// TIA Portal V21 export
DATA_BLOCK "LayoutPercorsi"   // DB2
{ S7_Optimized_Access := 'TRUE' }
// stored: MemoryReserve 100
   VAR
      PercorsoDa : Struct
         SerbatoioProdotto : Int := 5;
         PompaMono : Int := 5;
         ContropressioneUscitaMono : Int := 0;
         PompaPistoni : Int := 5;
         Sterilizzazione : Int := 5;
         RicicloLavoroASostatore : Int := 5;
         RicicloLavoroASottoRaffreddatore : Int := 0;
         Sostatore : Int := 5;
         Raffreddatore : Int := 5;
         IngressoAcidoCamiciaRaffreddatore : Int := 0;
         IngressoH20RaffreddamentoVersoMod : Int := 1;
         IngressoH20RaffreddamentoVersoSottoRaffredda : Int := 1;
         DevioAcidoCamiciaRaffreddatore : Int := 0;
         RitornoProdottoVersoValvolaVapInSterilizzazione : Int := 0;
         QCI : Int := 5;
         IngressoProdottoInVasca : Int := 5;
         IngressoProdottoInVascaDrenaggio : Int := 0;
         SorgenteAcqua : Int := 1;
         IngressoAcquaInVascaProdotto : Int := 0;
         IngressoAcquaInDivosfere : Int := 0;
         RitornoProdottoScartoVasca : Int := 0;
         RitornoProdottoScartoVascaDrenaggio : Int := 0;
         IngressoSodaAcido : Int := 0;
         DrenaggioIngressoSodaAcido : Int := 0;
         TankAcido : Int := 0;
         TankSoda : Int := 0;
         TuboAcidoSoda : Int := 0;
         PompaRicircolo : Int := 0;
         AlimentazionePompaCip : Int := 0;
         PompaCip : Int := 0;
         UscitaPompaCip : Int := 0;
         DrenaggioImpianto : Int := 0;
         DrenaggioVasca : Int := 0;
         "TronchettoPre-sterilizzazione" : Int := 5;
         SottoraffreddatoreARitornoProdotto : Int := 0;
         ReintegroH20Riscaldo : Int := 0;
         ModulanteRiscaldamentoAcqua : Int := 0;
         ScaricoCondense : Int := 0;
         AcquaCaldaAScaricoCondense : Int := 0;
         SorgenteVapore : Int := 6;
         VaporeInRiempimentoARicicloLavoro : Int := 0;
         RicicloLavoroASottoRaffreddatore_Vapore : Int := 0;
         RIempitriceMacropackCFT : Int := 0;
         ContropressioneADevioAcido : Int := 0;
         RitornoProdottoAControPressione : Int := 0;
         ScaricoVapInSterilizzazione : Int := 0;
         DevioAcidoARitornoProdotto : Int := 0;
         ValvolaManualeARitornoProdotto : Int := 0;
         RaffreddatoreAValvolaManuale : Int := 0;
         PompaRilancioTorri : Int := 1;
         PressurizzazioneSoda : Int := 0;
         PressurizzazioneAcido : Int := 0;
         IngressoVaporeSterilizzatore : Int := 0;
         AcquaCaldaAPompaRicircolo : Int := 0;
         ModulanteRaffreddamentoAcqua : Int := 1;
         IngressoRaffreddatore : Int := 1;
         EntrataSottoRaffreddatore : Int := 0;
         DrenaggioAcidoValvolaC : Int := 0;
         ValvolaX2aSottoraff : Int := 0;
      END_STRUCT;
      Visibilità : Struct
         PompaPistoni : Bool := FALSE;
      END_STRUCT;
   END_VAR
BEGIN
END_DATA_BLOCK
